Staubli VAL3: start.pgx

public program start()
begin

  prog:libLoad("Disk://XHS3023L/XHS3023L1")
  wait(taskStatus("loading")==-1)
  taskCreate "loading",10,loadNextOne("Disk://XHS3023L/XHS3023L2")
  call prog:start()

  prog:libLoad("Disk://XHS3023L/XHS3023L2")
  wait(taskStatus("loading")==-1)
  call prog:start()


end
